(* CoDeSys 2.3 export: E_BALLCOLOUR.EXP *)

(* Data type *)
TYPE E_BallColour :
(
	NoColour := 0,
	Yellow := 1,
	Blue := 2,
	Red := 3
);
END_TYPE
